SUBAPPLICATION Ventilsteuerung_Uebung_020c2 (* DigitalInput_I1 auf DigitalOutput_Q1; E_TON Einschaltverzögert; Zeit eingeben und speichern. *)
  (* Standard: 61499-2 *)
  (* Version 1.0, 2023-10-23, franz *)
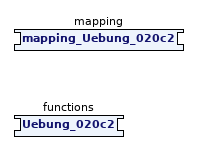
  SUBAPPS
    mapping : mapping_Uebung_020c2;
    functions : Uebung_020c2;
  END_SUBAPPS
END_SUBAPPLICATION
